Universal Robots URScript: T011_qwen2.5-coder_32b_baseline_rep1.urscript

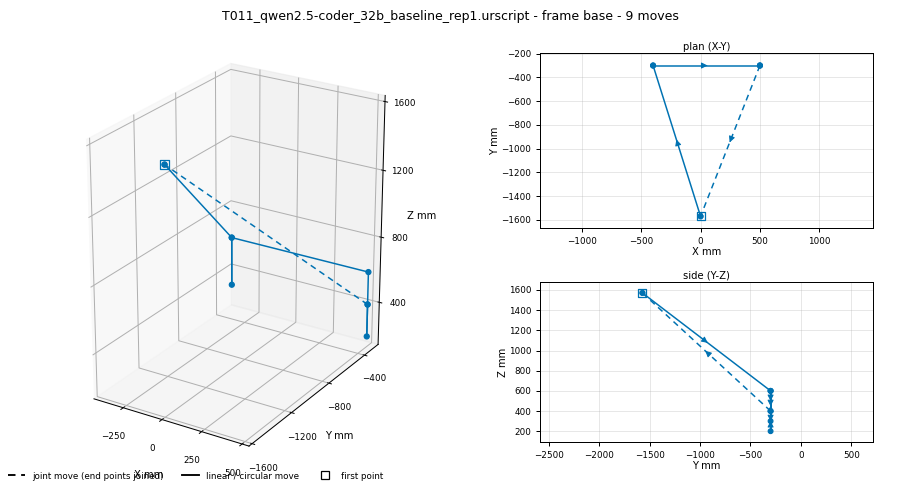
[picture p0: tool path of T011_qwen2.5-coder_32b_baseline_rep1.urscript in frame base, 9 of 9 moves have a stored position in this frame; points joined in program order, loops and branches not executed]
def dual_zone_pick_place():
    # Home position
    movej(p[0, -1.5708, 1.5708, -1.5708, -1.5708, 0], a=1.2, v=0.25)

    # Above storage bin
    movel(p[-0.4, -0.3, 0.6, 2.22, 2.22, 0], a=1.2, v=0.28)

    # Descend to pick
    movel(p[-0.4, -0.3, 0.3, 2.22, 2.22, 0], a=1.2, v=0.12)

    # Lift from bin
    movel(p[-0.4, -0.3, 0.6, 2.22, 2.22, 0], a=1.2, v=0.2)

    # Transit to handoff zone
    movel(p[0.5, -0.3, 0.6, 2.22, 2.22, 0], a=1.2, v=0.25)

    # Above handoff zone (additional move)
    movel(p[0.5, -0.3, 0.4, 2.22, 2.22, 0], a=1.2, v=0.28)

    # Descend to place
    movel(p[0.5, -0.3, 0.2, 2.22, 2.22, 0], a=1.2, v=0.12)

    # Lift from handoff zone (additional move)
    movel(p[0.5, -0.3, 0.4, 2.22, 2.22, 0], a=1.2, v=0.2)

    # Return to home position
    movej(p[0, -1.5708, 1.5708, -1.5708, -1.5708, 0], a=1.2, v=0.25)
end

dual_zone_pick_place()
